FUNCTION F_ResetExternalGroupError : BOOL
(**************************************************************************************
 * 	Application		:	BoxControl Framework
 *	Revision		:	$Revision: 404529 $
 *	Revision date	:	$Date: 2018-04-23 08:21:38 +0200 (Mo., 23 Apr 2018) $
 *	Last changed by	:	$Author: b7bolm $
 *	URL				:	$URL: http://almscdc.swisslog.com/repo/SWPD/Development/BoxControlFramework/20_Release/trunk/01_Software/BCF/BCF/JumpStart/20_Product/10_App/14_Groups/10_Lib/10_Conv/10_Functions/F_ResetExternalGroupError.TcPOU $
 *
 *	Purpose			:	Reset external error
 *						Add an External error, which will be reported over the configured
 *						position.
 *						
 *
 * ------------------------------------------------------------------------------------
 *	Copyright Swisslog [IP AG], Switzerland. All rights reserved.
 * 
 * ------------------------------------------------------------------------------------
 *	
 * 	Revision History: 
 *
 * 	VERSION			DATE			INITIALS			DESCRIPTION
 *	0.1				01.01.2001		swl					Example
 *
 **************************************************************************************)
VAR_INPUT
	eGroupNumber    : E_GroupNumber; 
	Reset			: BOOL;
END_VAR


// Validate inputs
IF eGroupNumber > E_GroupNumber.G_BEGIN_GROUP THEN
	IF __ISVALIDREF(GroupRegistry[eGroupNumber].rGroup) THEN
		// Reset external error on instance
		GroupRegistry[eGroupNumber].rGroup.M_ResetExternalError(
			mReset := Reset);
	END_IF
END_IF

END_FUNCTION

(* stored: Version 1.1.0.1, ProductVersion 3.1.4022.12
   POU F_ResetExternalGroupError: Id {623c1e55-432e-4df9-8d78-24b562cc8867}, SpecialFunc None *)
